//{attribute 'strict'}
TYPE E_SYSTEM_AutomationMode :
(
	E_SYSTEM_EXTERNAL		:= 0,
	E_SYSTEM_CML			:= 1,
	E_SYSTEM_LARS			:= 2,
	E_SYSTEM_SIDEFLEX		:= 3

);
END_TYPE

(* stored: Version 1.1.0.1
   DUT E_SYSTEM_AutomationMode: Id {dc210746-b6b6-48c2-b669-37065675dec5} *)
